# EPICS autosave request: iocBoot/iocsnd/snd.req
## Records to be saved by autosave
$(BL):$(DEV):$(GROUP):Threshold
$(BL):$(DEV):$(GROUP):reference.DESC
